FUNCTION_BLOCK FB_TelescopeState IMPLEMENTS I_TelescopeState
VAR_INPUT
END_VAR
VAR_OUTPUT
END_VAR
VAR
	pMachine 		: POINTER TO FB_TelescopeMachine;
	comm			: I_Comm;
	bMainReset		: BOOL;	// Used to reset each state if a state change happens before completion
	bInitialize		: BOOL;
	bPark			: BOOL;
	bReset			: BOOL;
	bSlew			: BOOL;
	bStop			: BOOL;
	bTrack			: BOOL;
	bError			: BOOL;
	iStage			: UINT;
END_VAR

METHOD Error : BOOL
VAR_INPUT
END_VAR
bMainReset := TRUE;
pMachine^.eState.Main();
bMainReset := FALSE;
pMachine^.eState := E_TelescopeState.error;
END_METHOD

METHOD FB_init : BOOL
VAR_INPUT
	bInitRetains 	: BOOL; // if TRUE, the retain variables are initialized (warm start / cold start)
	bInCopyCode 	: BOOL;  // if TRUE, the instance afterwards gets moved into the copy code (online change)
	pMachine 		: POINTER TO FB_TelescopeMachine;
	comm			: I_Comm;
END_VAR
THIS^.pMachine := pMachine;
THIS^.comm := comm;
END_METHOD

METHOD Initialize : BOOL
VAR_INPUT
END_VAR
IF NOT pMachine^.pControl^.bError AND pMachine^.eState = E_TelescopeState.parked THEN
	pMachine^.eState := E_TelescopeState.initializing;
END_IF
END_METHOD

METHOD Main : BOOL
VAR_INPUT
END_VAR
END_METHOD

METHOD Park : BOOL
VAR_INPUT
END_VAR
IF NOT pMachine^.pControl^.bError AND pMachine^.pControl^.bPower  THEN
	bMainReset := TRUE;
	pMachine^.eState.Main();
	bMainReset := FALSE;
	pMachine^.eState := E_TelescopeState.parking;
END_IF
END_METHOD

METHOD Reset : BOOL
VAR_INPUT
END_VAR
bReset := TRUE;
END_METHOD

METHOD Slew : BOOL
VAR_INPUT
END_VAR
IF NOT pMachine^.pControl^.bError AND pMachine^.pControl^.bPower  THEN
	bMainReset := TRUE;
	pMachine^.eState.Main();
	bMainReset := FALSE;
	pMachine^.eState := E_TelescopeState.slewing;
END_IF
END_METHOD

METHOD Stop : BOOL
VAR_INPUT
END_VAR
IF NOT pMachine^.pControl^.bError THEN
	bMainReset := TRUE;
	pMachine^.eState.Main();
	bMainReset := FALSE;
	pMachine^.eState := E_TelescopeState.stopping;
END_IF
END_METHOD

METHOD Track : BOOL
VAR_INPUT
END_VAR
IF NOT pMachine^.pControl^.bError AND pMachine^.pControl^.bPower  THEN
	bMainReset := TRUE;
	pMachine^.eState.Main();
	bMainReset := FALSE;
	pMachine^.eState := E_TelescopeState.tracking;
END_IF
END_METHOD

END_FUNCTION_BLOCK

(* stored: Version 1.1.0.1, ProductVersion 3.1.4024.15
   POU FB_TelescopeState: Id {a1655b2a-b366-4c97-b1c5-df3d2b5e068d}, SpecialFunc None
   Method Error: Id {e8b11311-e16b-4c9b-82ce-52a1c79b8cc6}
   Method FB_init: Id {939ce836-b748-4327-8af4-fef7b1a3e467}
   Method Initialize: Id {4014e65c-f049-46d7-ab38-f9d8532488b1}
   Method Main: Id {eab1ce7f-ef78-48ef-ab88-bd1f860b5b79}
   Method Park: Id {1d7b2094-1b9e-4f3f-8684-35da700e0b9a}
   Method Reset: Id {57d7d305-bed4-400e-bbf9-c181dc7d793e}
   Method Slew: Id {e5dd4f78-c7c2-4163-9dee-c9e4a43c707b}
   Method Stop: Id {f88b6084-031f-4751-912f-ee2fd3d7f783}
   Method Track: Id {33662814-9536-4e5d-81b1-cbf07479cb1d} *)
